{attribute 'qualified_only' := ''}
{attribute 'strict' := ''}
TYPE E_ConveyorLevelerState :
(
	STOP := 0,
	HOME_FAST_SEARCH := 10,
	HOME_SLOW_EXIT_SENSOR := 11,
	HOME_SET_ENCODER := 12,
	MANUAL := 20,
	AUTO_LEVELING := 30,
	FAULT := 40
);
END_TYPE

(* stored: Version 1.1.0.1
   DUT E_ConveyorLevelerState: Id {0466d059-145d-4d3c-86a3-b95ea53ad822} *)
